# EPICS substitutions: TS02K-MO-IOC-01App/Db/TS02K-MO-IOC-01_expanded.substitutions
# This file was automatically generated on Wed 19 Aug 2026 15:11:30 BST from
# source: /scratch/ronaldo/id1051/IDLAB-BUILDER/etc/makeIocs/TS16K-MO-IOC-01.xml
#
# *** Please do not edit this file: edit the source file instead. ***
#

# Macros:
#  IOC  Device prefix
file $(IOCSTATS)/db/iocAdminSoft.db
{
pattern { IOC }
    { "TS21K-MO-IOC-01" }
}

# Macros:
#  IOC  Device prefix
file $(IOCSTATS)/db/iocAdminScanMon.db
{
pattern { IOC }
    { "TS21K-MO-IOC-01" }
}

# Macros:
#  PORT      The asyn port for the pmac controller
#  P         PV Prefix
#  NAXES     Number of axes
#  TIMEOUT   Timeout for controller communication
#  FEEDRATE  feedrate below which we go into error
#  CSG0      Name for Coordinate System Group 0
#  CSG1      Name for Coordinate System Group 1
#  CSG2      Name for Coordinate System Group 2
#  CSG3      Name for Coordinate System Group 3
#  CSG4      Name for Coordinate System Group 4
#  CSG5      Name for Coordinate System Group 5
#  CSG6      Name for Coordinate System Group 6
#  CSG7      Name for Coordinate System Group 7
file $(PMAC)/db/pmacController.template
{
pattern { PORT, P, NAXES, TIMEOUT, FEEDRATE, CSG0, CSG1, CSG2, CSG3, CSG4, CSG5, CSG6, CSG7 }
    { "pwbrick", "TS21K-MO-SERVO-01", "8", "4", "100", "", "", "", "", "", "", "", "" }
}

# Macros:
#  PORT  The asyn port for the pmac controller
#  P     PV Prefix
file $(PMAC)/db/powerPmacStatus.template
{
pattern { PORT, P }
    { "pwbrick", "TS21K-MO-SERVO-01" }
}

# Macros:
#  PMAC  Pmac/Geobrick name
#  AXIS  Axis number
#  PORT  Asyn port
file $(PMAC)/db/pmacStatusAxis.template
{
pattern { PMAC, AXIS, PORT }
    { "TS21K-MO-SERVO-01", "1", "pwbrick" }
    { "TS21K-MO-SERVO-01", "2", "pwbrick" }
    { "TS21K-MO-SERVO-01", "3", "pwbrick" }
    { "TS21K-MO-SERVO-01", "4", "pwbrick" }
}

# Macros:
#  PORT        The asyn port for the pmac cs controller
#  PARENTPORT  The asyn port for the parent pmac controller
#  PMAC        PV Prefix for the motor controller
#  CS          Coordinate System Number for the cs controller
#  TIMEOUT     Timeout for controller communication
file $(PMAC)/db/pmacCsController.template
{
pattern { PORT, PARENTPORT, PMAC, CS, TIMEOUT }
    { "PPMAC_1_CS_2", "pwbrick", "TS21K-MO-SERVO-01", "2", "4" }
    { "PPMAC_1_CS_3", "pwbrick", "TS21K-MO-SERVO-01", "3", "4" }
}

# Macros:
#  P                Device Prefix
#  M                Device Suffix
#  PORT             Delta tau motor controller
#  ADDR             Address on controller
#  DESC             Description, displayed on EDM screen
#  MRES             Motor Step Size (EGU)
#  VELO             Velocity (EGU/s)
#  PREC             Display Precision
#  EGU              Engineering Units
#  TWV              Tweak Step Size (EGU)
#  DTYP             DTYP of record
#  DIR              User Direction
#  VBAS             Base Velocity (EGU/s)
#  VMAX             Max Velocity (EGU/s), defaults to VELO
#  ACCL             Seconds to Velocity
#  BDST             BL Distance (EGU)
#  BVEL             BL Velocity (EGU/s)
#  BACC             BL Seconds to Veloc.
#  DHLM             Dial High Limit
#  DLLM             Dial Low Limit
#  HLM              User High Limit
#  LLM              User Low Limit
#  HLSV             HW Lim. Violation Svr
#  INIT             Startup commands
#  SREV             Steps per Revolution
#  RRES             Readback Step Size (EGU)
#  ERES             Encoder Step Size (EGU)
#  JAR              Jog Acceleration (EGU/s^2)
#  UEIP             Use Encoder If Present
#  URIP             Use RDBL If Present
#  RDBL             Readback Location, set URIP = 1 if you specify this
#  RLNK             Readback output link
#  RTRY             Max retry count
#  DLY              Readback settle time (s)
#  OFF              User Offset (EGU)
#  RDBD             Retry Deadband (EGU)
#  FOFF             Freeze Offset, 0=variable, 1=frozen
#  ADEL             Alarm monitor deadband (EGU)
#  NTM              New Target Monitor, only set to 0 for soft motors
#  FEHIGH           HIGH limit for following error
#  FEHIHI           HIHI limit for following error
#  FEHHSV           HIHI alarm severity for following error
#  FEHSV            HIGH alarm severity for following error
#  SCALE            Scale factor, if pmacSetAxisScale is used this should be set
#  HOMEVIS          If 1 then home is visible on the gui
#  HOMEVISSTR       If HOMEVIS=0, then display this text on the gui instead
#  name             Object name and gui association name
#  alh              Set this to alh to add the motor to the alarm handler and send emails,
#  gda_name         Name to export this as to GDA
#  gda_desc         Description to export this as to GDA
#  SPORT            Delta tau motor controller comms port
#  HOME             Prefix for autohome instance. Defaults to $(P). If unspecified,
#  ALLOW_HOMED_SET  Set to a blank to allow this axis to have its homed
file $(PMAC)/db/dls_pmac_asyn_motor.template
{
pattern { P, M, PORT, ADDR, DESC, MRES, VELO, PREC, EGU, TWV, DTYP, DIR, VBAS, VMAX, ACCL, BDST, BVEL, BACC, DHLM, DLLM, HLM, LLM, HLSV, INIT, SREV, RRES, ERES, JAR, UEIP, URIP, RDBL, RLNK, RTRY, DLY, OFF, RDBD, FOFF, ADEL, NTM, FEHIGH, FEHIHI, FEHHSV, FEHSV, SCALE, HOMEVIS, HOMEVISSTR, name, alh, gda_name, gda_desc, SPORT, HOME, PMAC, ALLOW_HOMED_SET }
    { "TS21K-MO-SERVO-01", ":MOT", "pwbrick", "1", "Gap U/S", "0.000005", "1", "6", "mm", "0.01", "asynMotor", "0", "0", "$(VELO)", "0.5", "0", "0", "", "89.165825", "54.965825", "", "", "MAJOR", "", "1000", "", "", "", "0", "0", "", "", "0", "0", "-70.35573", "", "0", "0", "1", "0", "0", "NO_ALARM", "NO_ALARM", "1", "1", "Use motor summary screen", "IDGUI.servo.01", "None", "", "$(DESC)", "SSHP", "$(P)", "TS21K-MO-SERVO-01", "#" }
    { "TS21K-MO-SERVO-02", ":MOT", "pwbrick", "2", "Gap D/S", "0.000005", "1", "6", "mm", "0.01", "asynMotor", "0", "0", "$(VELO)", "0.5", "0", "0", "", "88.542205", "54.342205", "", "", "MAJOR", "", "1000", "", "", "", "0", "0", "", "", "0", "0", "-69.257395", "", "0", "0", "1", "0", "0", "NO_ALARM", "NO_ALARM", "1", "1", "Use motor summary screen", "IDGUI.servo.02", "None", "", "$(DESC)", "SSHP", "$(P)", "TS21K-MO-SERVO-01", "#" }
    { "TS21K-MO-SERVO-03", ":MOT", "pwbrick", "3", "Offset U/S", "0.000005", "0.1", "6", "mm", "0.01", "asynMotor", "0", "0", "$(VELO)", "0.5", "0", "0", "", "47.5956", "46.7256", "", "", "MAJOR", "", "1000", "", "", "", "0", "0", "", "", "0", "0", "-47.857515", "", "0", "0", "1", "0", "0", "NO_ALARM", "NO_ALARM", "1", "1", "Use motor summary screen", "IDGUI.servo.03", "None", "", "$(DESC)", "SSHP", "$(P)", "TS21K-MO-SERVO-01", "#" }
    { "TS21K-MO-SERVO-04", ":MOT", "pwbrick", "4", "Offset D/S", "0.000005", "0.1", "6", "mm", "0.01", "asynMotor", "0", "0", "$(VELO)", "0.5", "0", "0", "", "47.246615", "46.376615", "", "", "MAJOR", "", "1000", "", "", "", "0", "0", "", "", "0", "0", "-47.216195", "", "0", "0", "1", "0", "0", "NO_ALARM", "NO_ALARM", "1", "1", "Use motor summary screen", "IDGUI.servo.04", "None", "", "$(DESC)", "SSHP", "$(P)", "TS21K-MO-SERVO-01", "#" }
}

# Macros:
#  P           Device Prefix
#  M           Device Suffix
#  PORT        Coordinate System object that this motor belongs to
#  ADDR        Address on controller
#  DESC        Description, displayed on EDM screen
#  MRES        Motor Step Size (EGU)
#  VELO        Velocity (EGU/s)
#  PREC        Display Precision
#  EGU         Engineering Units
#  TWV         Tweak Step Size (EGU)
#  DTYP        DTYP of record
#  DIR         User Direction
#  VBAS        Base Velocity (EGU/s)
#  VMAX        Max Velocity (EGU/s), defaults to VELO
#  ACCL        Seconds to Velocity
#  BDST        BL Distance (EGU)
#  BVEL        BL Velocity (EGU/s)
#  BACC        BL Seconds to Veloc.
#  DHLM        Dial High Limit
#  DLLM        Dial Low Limit
#  HLM         User High Limit
#  LLM         User Low Limit
#  HLSV        HW Lim. Violation Svr
#  INIT        Startup commands
#  SREV        Steps per Revolution
#  RRES        Readback Step Size (EGU)
#  ERES        Encoder Step Size (EGU)
#  JAR         Jog Acceleration (EGU/s^2)
#  UEIP        Use Encoder If Present
#  URIP        Use RDBL If Present
#  RDBL        Readback Location, set URIP = 1 if you specify this
#  RLNK        Readback output link
#  RTRY        Max retry count
#  DLY         Readback settle time (s)
#  OFF         User Offset (EGU)
#  RDBD        Retry Deadband (EGU)
#  FOFF        Freeze Offset, 0=variable, 1=frozen
#  ADEL        Alarm monitor deadband (EGU)
#  NTM         New Target Monitor, only set to 0 for soft motors
#  FEHIGH      HIGH limit for following error
#  FEHIHI      HIHI limit for following error
#  FEHHSV      HIHI alarm severity for following error
#  FEHSV       HIGH alarm severity for following error
#  SCALE       Scale factor, if pmacSetAxisScale is used this should be set
#  HOMEVIS     If 1 then home is visible on the gui
#  HOMEVISSTR  If HOMEVIS=0, then display this text on the gui instead
#  name        Object name and gui association name
#  alh         Set this to alh to add the motor to the alarm handler and send emails,
#  gda_name    Name to export this as to GDA
#  gda_desc    Description to export this as to GDA
file $(PMAC)/db/dls_pmac_cs_asyn_motor.template
{
pattern { P, M, PORT, ADDR, DESC, MRES, VELO, PREC, EGU, TWV, DTYP, DIR, VBAS, VMAX, ACCL, BDST, BVEL, BACC, DHLM, DLLM, HLM, LLM, HLSV, INIT, SREV, RRES, ERES, JAR, UEIP, URIP, RDBL, RLNK, RTRY, DLY, OFF, RDBD, FOFF, ADEL, NTM, FEHIGH, FEHIHI, FEHHSV, FEHSV, SCALE, HOMEVIS, HOMEVISSTR, name, alh, gda_name, gda_desc, PMAC, CS }
    { "TS21K-MO-SERVC-01:CS", ":GAP", "PPMAC_1_CS_2", "1", "ID Gap", "0.0001", "1", "5", "mm", "0.02", "asynMotor", "0", "0", "$(VELO)", "0.5", "0", "0", "", "36.8", "2.6", "", "", "MAJOR", "", "1000", "", "", "", "0", "0", "", "", "0", "0", "0", "", "0", "0", "1", "0", "0", "NO_ALARM", "NO_ALARM", "1", "1", "Use motor summary screen", "IDGAP", "None", "", "$(DESC)", "TS21K-MO-SERVO-01", "2" }
    { "TS21K-MO-SERVC-01:CS", ":OFFSET", "PPMAC_1_CS_3", "1", "ID Offset", "0.0001", "0.1", "5", "mm", "0.02", "asynMotor", "0", "0", "$(VELO)", "0.5", "0", "0", "", "0.32", "-0.55", "", "", "MAJOR", "", "1000", "", "", "", "0", "0", "", "", "0", "0", "0", "", "0", "0", "1", "0", "0", "NO_ALARM", "NO_ALARM", "1", "1", "Use motor summary screen", "IDOFFSET", "None", "", "$(DESC)", "TS21K-MO-SERVO-01", "3" }
}

# Macros:
#  name    name for gui element
#  idname  name for gui screen (do not include spaces)
#  server  linux server to use to bridge through to for pmac control
#  pmac    name of pmac controller
#  dom     first part of prefix, used to build gui macros
#  suff1   always zero - c.f. jira ID-739
file $(IDMOTION)/db/IDM_gui.template
{
pattern { name, idname, server, pmac, dom, suff1 }
    { "MOTION", "HPMU-K21", "hpmu-k21", "192.168.121.1", "TS21K", "0" }
}

# Macros:
#  prefix  record prefix
#  port    powerbrick asyn port from pmacCreateController invocation
#  name    gui element
file $(IDMOTION)/db/IDM_encSync.template
{
pattern { prefix, port, name }
    { "TS21K-MO-PMAC-01", "pwbrick", "IDGUI.ENCSYNC" }
}

file $(IDMOTION)/db/IDM_ampLoss.template
{
pattern {prefix, port}
    { "TS21K-MO-PMAC-01", "pwbrick" }
}

# Macros:
#  prefix  record prefix
#  port    powerbrick asyn port from pmacCreateController invocation
#  name    gui element
file $(IDMOTION)/db/IDM_stop.template
{
pattern { prefix, port, name }
    { "TS21K-MO-PMAC-01", "pwbrick", "IDGUI.STOP" }
}

# Macros:
#  prefix  pv prefix e.g. TS02K-MO-
#  name    Template argument
file $(IDMOTION)/db/IDM_defer.template
{
pattern { prefix, name }
    { "TS21K-MO-", "IDGUI.DEFER" }
}

# Macros:
#  prefix  pv prefix e.g. TS02K-MO-
file $(IDMOTION)/db/IDM_gap.template
{
pattern { prefix }
    { "TS21K-MO-" }
}

# Macros:
#  prefix  pv prefix e.g. TS02K-MO-
file $(IDMOTION)/db/IDM_single.template
{
pattern { prefix }
    { "TS21K-MO-" }
}

# Macros:
#  prefix  pv prefix, e.g. SR02J-MO-
#  axx     axis number e.g. 01, 02, etc
file $(IDMOTION)/db/IDM_lim.template
{
pattern { prefix, axx }
    { "TS21K-MO-", "01" }
    { "TS21K-MO-", "02" }
    { "TS21K-MO-", "03" }
    { "TS21K-MO-", "04" }
}

# Macros:
#  prefix  pv prefix, e.g. SR02J-MO-
#  axx     axis number e.g. 01, 02, etc
file $(IDMOTION)/db/IDM_posok.template
{
pattern { prefix, axx }
    { "TS21K-MO-", "01" }
    { "TS21K-MO-", "02" }
    { "TS21K-MO-", "03" }
    { "TS21K-MO-", "04" }
}

# Macros:
#  name    gui component name
#  prefix  device prefix
#  idname  name for insertion device
file $(IDPLC)/db/idplc_gui.template
{
pattern { name, prefix, idname }
    { "IDGUI.PLC", "TS21K-MO", "HPMU-K21" }
}
